(* IEC 61131-3 sources: rtacc/examples/XOR, 1 file *)

(* ---- XOR.st ---- *)
FUNCTION XOR_FUNC : BOOL
VAR_INPUT
    A : BOOL;
    B : BOOL;
END_VAR

XOR_FUNC := A XOR B;

END_FUNCTION
